FUNCTION CompareDate : int
VAR_INPUT
	timestruct1 : TIMESTRUCT;
	timestruct2 : TIMESTRUCT;
	
END_VAR
VAR
END_VAR

IF timestruct1.wYear < timestruct2.wYear THEN
	CompareDate := -10;
ELSIF timestruct1.wYear > timestruct2.wYear THEN
		CompareDate := 10;
ELSE 
	IF timestruct1.wMonth < timestruct2.wMonth THEN
		CompareDate := -10;
	ELSIF  timestruct1.wMonth > timestruct2.wMonth THEN
				CompareDate := 10;
	ELSE
		IF timestruct1.wDay < timestruct2.wDay THEN
			CompareDate := -10;
		ELSIF timestruct1.wDay > timestruct2.wDay THEN
			CompareDate := 10;
		ELSE 
			CompareDate := 0;
		END_IF

	END_IF
END_IF

END_FUNCTION

(* stored: Version 1.1.0.1, ProductVersion 3.1.4024.12
   POU CompareDate: Id {f69f33fe-160c-4f83-bb16-a221e7432766}, SpecialFunc None *)
